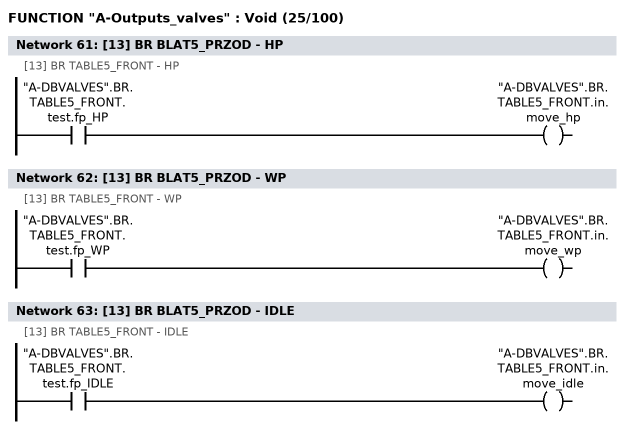
      O "A-DBVALVES".BR.TABLE5_FRONT.test.fp_HP;
//    O     "A-Flags".STATION.IN_HP_STEP
      = "A-DBVALVES".BR.TABLE5_FRONT.in.move_hp;
NETWORK
TITLE = [13] BR BLAT5_PRZOD - WP
//[13] BR TABLE5_FRONT - WP
      O "A-DBVALVES".BR.TABLE5_FRONT.test.fp_WP;
      = "A-DBVALVES".BR.TABLE5_FRONT.in.move_wp;
NETWORK
TITLE = [13] BR BLAT5_PRZOD - IDLE
//[13] BR TABLE5_FRONT - IDLE
      O "A-DBVALVES".BR.TABLE5_FRONT.test.fp_IDLE;
      = "A-DBVALVES".BR.TABLE5_FRONT.in.move_idle;
NETWORK
TITLE = [13] BR BLAT5_PRZOD
//[13] BR TABLE5_FRONT
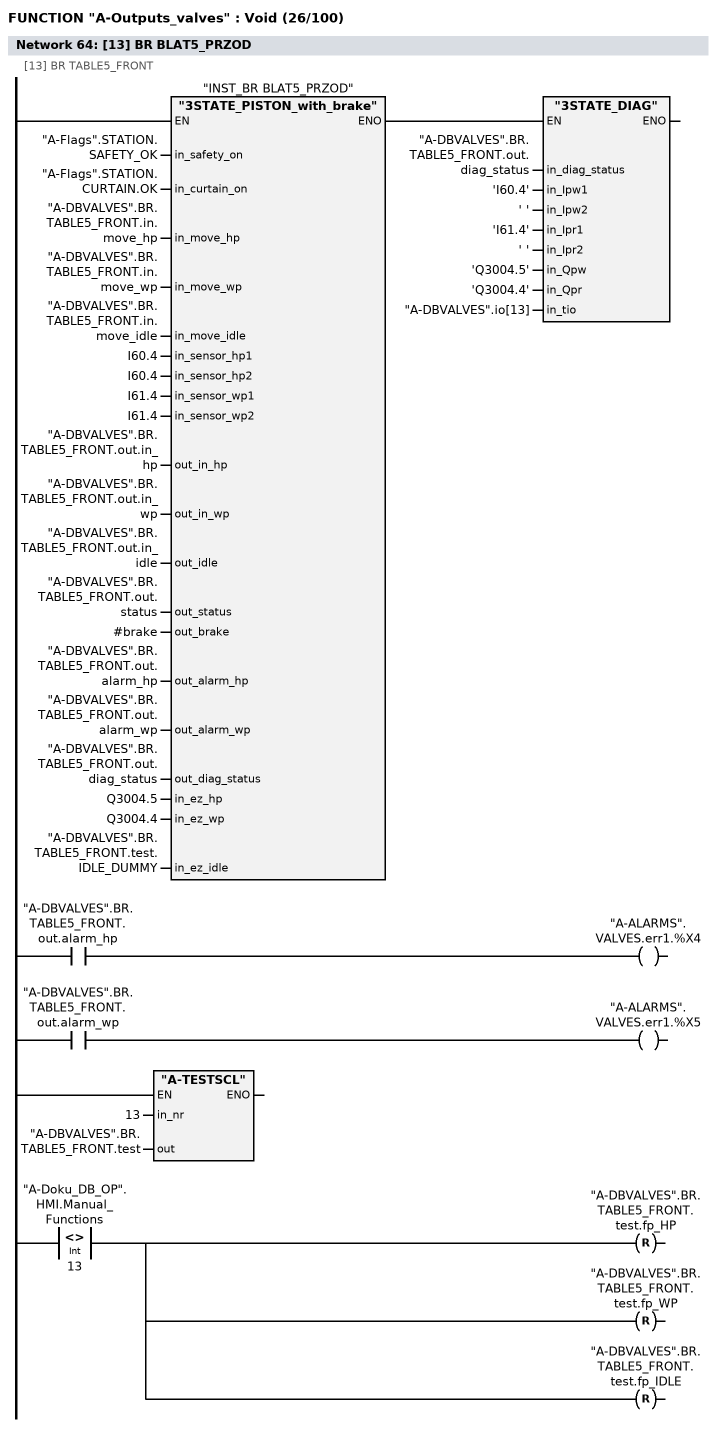
      CALL "3STATE_PISTON_with_brake", "INST_BR BLAT5_PRZOD"
      (  in_safety_on                := "A-Flags".STATION.SAFETY_OK ,
         in_curtain_on               := "A-Flags".STATION.CURTAIN.OK ,
         in_move_hp                  := "A-DBVALVES".BR.TABLE5_FRONT.in.move_hp ,
         in_move_wp                  := "A-DBVALVES".BR.TABLE5_FRONT.in.move_wp ,
         in_move_idle                := "A-DBVALVES".BR.TABLE5_FRONT.in.move_idle ,
         in_sensor_hp1               := I60.4 ,
         in_sensor_hp2               := I60.4 ,
         in_sensor_wp1               := I61.4 ,
         in_sensor_wp2               := I61.4 ,
         out_in_hp                   := "A-DBVALVES".BR.TABLE5_FRONT.out.in_hp ,
         out_in_wp                   := "A-DBVALVES".BR.TABLE5_FRONT.out.in_wp ,
         out_idle                    := "A-DBVALVES".BR.TABLE5_FRONT.out.in_idle ,
         out_status                  := "A-DBVALVES".BR.TABLE5_FRONT.out.status ,
         out_brake                   := #brake ,
         out_alarm_hp                := "A-DBVALVES".BR.TABLE5_FRONT.out.alarm_hp ,
         out_alarm_wp                := "A-DBVALVES".BR.TABLE5_FRONT.out.alarm_wp ,
         out_diag_status             := "A-DBVALVES".BR.TABLE5_FRONT.out.diag_status ,
         in_ez_hp                    := Q3004.5 ,
         in_ez_wp                    := Q3004.4 ,
         in_ez_idle                  := "A-DBVALVES".BR.TABLE5_FRONT.test.IDLE_DUMMY
      );

      CALL "3STATE_DIAG"
      (  in_diag_status              := "A-DBVALVES".BR.TABLE5_FRONT.out.diag_status ,
         in_Ipw1                     := 'I60.4' ,
         in_Ipw2                     := ' ' ,
         in_Ipr1                     := 'I61.4' ,
         in_Ipr2                     := ' ' ,
         in_Qpw                      := 'Q3004.5' ,
         in_Qpr                      := 'Q3004.4' ,
         in_tio                      := "A-DBVALVES".io[13]
      );

      A "A-DBVALVES".BR.TABLE5_FRONT.out.alarm_hp;
      = "A-ALARMS".VALVES.err1.%X4;

      A "A-DBVALVES".BR.TABLE5_FRONT.out.alarm_wp;
      = "A-ALARMS".VALVES.err1.%X5;

      CALL "A-TESTSCL"
      (  in_nr                       := 13 ,
         out                         := "A-DBVALVES".BR.TABLE5_FRONT.test
      );

      A(;
      L "A-Doku_DB_OP".HMI.Manual_Functions;
      L 13;
      <>I;
      );
      R "A-DBVALVES".BR.TABLE5_FRONT.test.fp_HP;
      R "A-DBVALVES".BR.TABLE5_FRONT.test.fp_WP;
      R "A-DBVALVES".BR.TABLE5_FRONT.test.fp_IDLE;
NETWORK
TITLE = -

NETWORK
TITLE = [14] BR BLAT_TYL_LEWY - HP
//[14] BR TABLE_REAR_LEFT - HP
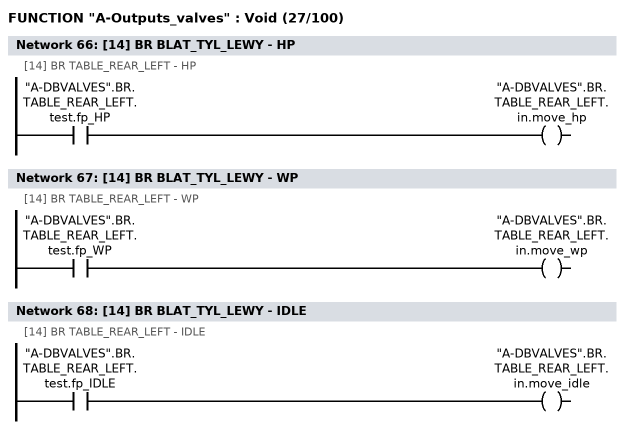
      O "A-DBVALVES".BR.TABLE_REAR_LEFT.test.fp_HP;
//    O     "A-Flags".STATION.IN_HP_STEP
      = "A-DBVALVES".BR.TABLE_REAR_LEFT.in.move_hp;
NETWORK
TITLE = [14] BR BLAT_TYL_LEWY - WP
//[14] BR TABLE_REAR_LEFT - WP
      O "A-DBVALVES".BR.TABLE_REAR_LEFT.test.fp_WP;
      = "A-DBVALVES".BR.TABLE_REAR_LEFT.in.move_wp;
NETWORK
TITLE = [14] BR BLAT_TYL_LEWY - IDLE
//[14] BR TABLE_REAR_LEFT - IDLE
      O "A-DBVALVES".BR.TABLE_REAR_LEFT.test.fp_IDLE;
      = "A-DBVALVES".BR.TABLE_REAR_LEFT.in.move_idle;
NETWORK
TITLE = [14] BR BLAT_TYL_LEWY
//[14] BR TABLE_REAR_LEFT
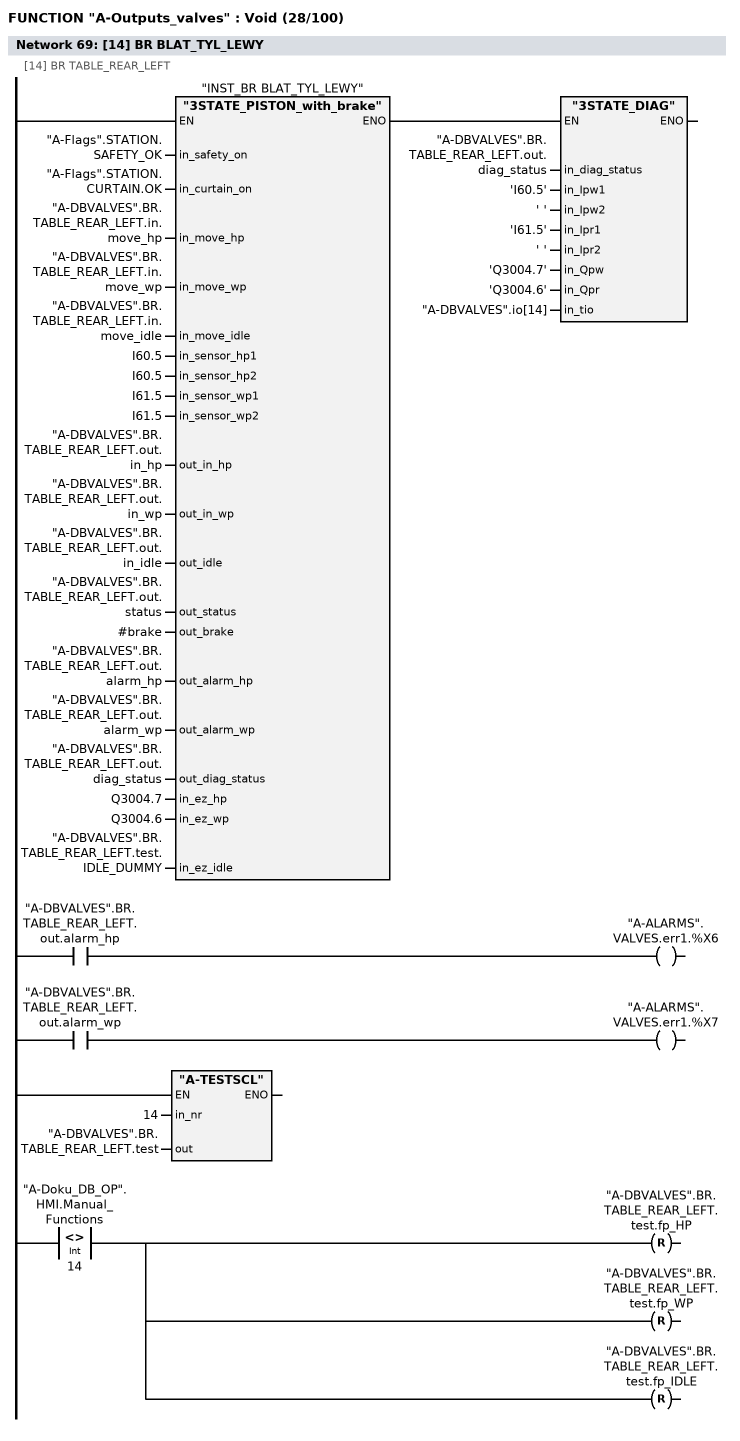
      CALL "3STATE_PISTON_with_brake", "INST_BR BLAT_TYL_LEWY"
      (  in_safety_on                := "A-Flags".STATION.SAFETY_OK ,
         in_curtain_on               := "A-Flags".STATION.CURTAIN.OK ,
         in_move_hp                  := "A-DBVALVES".BR.TABLE_REAR_LEFT.in.move_hp ,
         in_move_wp                  := "A-DBVALVES".BR.TABLE_REAR_LEFT.in.move_wp ,
         in_move_idle                := "A-DBVALVES".BR.TABLE_REAR_LEFT.in.move_idle ,
         in_sensor_hp1               := I60.5 ,
         in_sensor_hp2               := I60.5 ,
         in_sensor_wp1               := I61.5 ,
         in_sensor_wp2               := I61.5 ,
         out_in_hp                   := "A-DBVALVES".BR.TABLE_REAR_LEFT.out.in_hp ,
         out_in_wp                   := "A-DBVALVES".BR.TABLE_REAR_LEFT.out.in_wp ,
         out_idle                    := "A-DBVALVES".BR.TABLE_REAR_LEFT.out.in_idle ,
         out_status                  := "A-DBVALVES".BR.TABLE_REAR_LEFT.out.status ,
         out_brake                   := #brake ,
         out_alarm_hp                := "A-DBVALVES".BR.TABLE_REAR_LEFT.out.alarm_hp ,
         out_alarm_wp                := "A-DBVALVES".BR.TABLE_REAR_LEFT.out.alarm_wp ,
         out_diag_status             := "A-DBVALVES".BR.TABLE_REAR_LEFT.out.diag_status ,
         in_ez_hp                    := Q3004.7 ,
         in_ez_wp                    := Q3004.6 ,
         in_ez_idle                  := "A-DBVALVES".BR.TABLE_REAR_LEFT.test.IDLE_DUMMY
      );

      CALL "3STATE_DIAG"
      (  in_diag_status              := "A-DBVALVES".BR.TABLE_REAR_LEFT.out.diag_status ,
         in_Ipw1                     := 'I60.5' ,
         in_Ipw2                     := ' ' ,
         in_Ipr1                     := 'I61.5' ,
         in_Ipr2                     := ' ' ,
         in_Qpw                      := 'Q3004.7' ,
         in_Qpr                      := 'Q3004.6' ,
         in_tio                      := "A-DBVALVES".io[14]
      );

      A "A-DBVALVES".BR.TABLE_REAR_LEFT.out.alarm_hp;
      = "A-ALARMS".VALVES.err1.%X6;

      A "A-DBVALVES".BR.TABLE_REAR_LEFT.out.alarm_wp;
      = "A-ALARMS".VALVES.err1.%X7;

      CALL "A-TESTSCL"
      (  in_nr                       := 14 ,
         out                         := "A-DBVALVES".BR.TABLE_REAR_LEFT.test
      );

      A(;
      L "A-Doku_DB_OP".HMI.Manual_Functions;
      L 14;
      <>I;
      );
      R "A-DBVALVES".BR.TABLE_REAR_LEFT.test.fp_HP;
      R "A-DBVALVES".BR.TABLE_REAR_LEFT.test.fp_WP;
      R "A-DBVALVES".BR.TABLE_REAR_LEFT.test.fp_IDLE;
NETWORK
TITLE = -

NETWORK
TITLE = [15] BR BLAT_TYL_PRAWY - HP
//[15] BR TABLE_REAR_RIGHT - HP
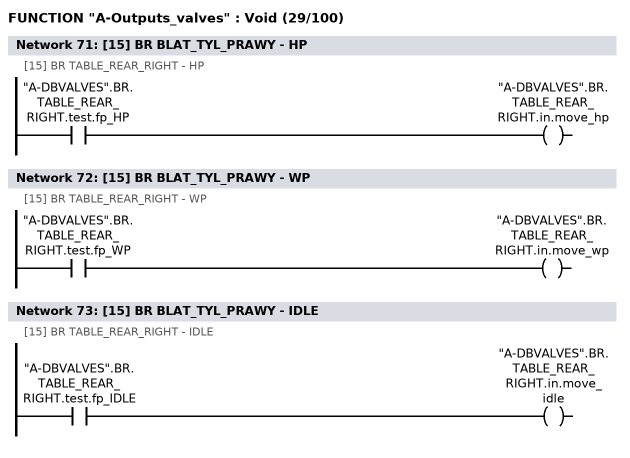
      O "A-DBVALVES".BR.TABLE_REAR_RIGHT.test.fp_HP;
//    O     "A-Flags".STATION.IN_HP_STEP
      = "A-DBVALVES".BR.TABLE_REAR_RIGHT.in.move_hp;
NETWORK
TITLE = [15] BR BLAT_TYL_PRAWY - WP
//[15] BR TABLE_REAR_RIGHT - WP
      O "A-DBVALVES".BR.TABLE_REAR_RIGHT.test.fp_WP;
      = "A-DBVALVES".BR.TABLE_REAR_RIGHT.in.move_wp;
NETWORK
TITLE = [15] BR BLAT_TYL_PRAWY - IDLE
//[15] BR TABLE_REAR_RIGHT - IDLE
      O "A-DBVALVES".BR.TABLE_REAR_RIGHT.test.fp_IDLE;
      = "A-DBVALVES".BR.TABLE_REAR_RIGHT.in.move_idle;
NETWORK
TITLE = [15] BR BLAT_TYL_PRAWY
//[15] BR TABLE_REAR_RIGHT
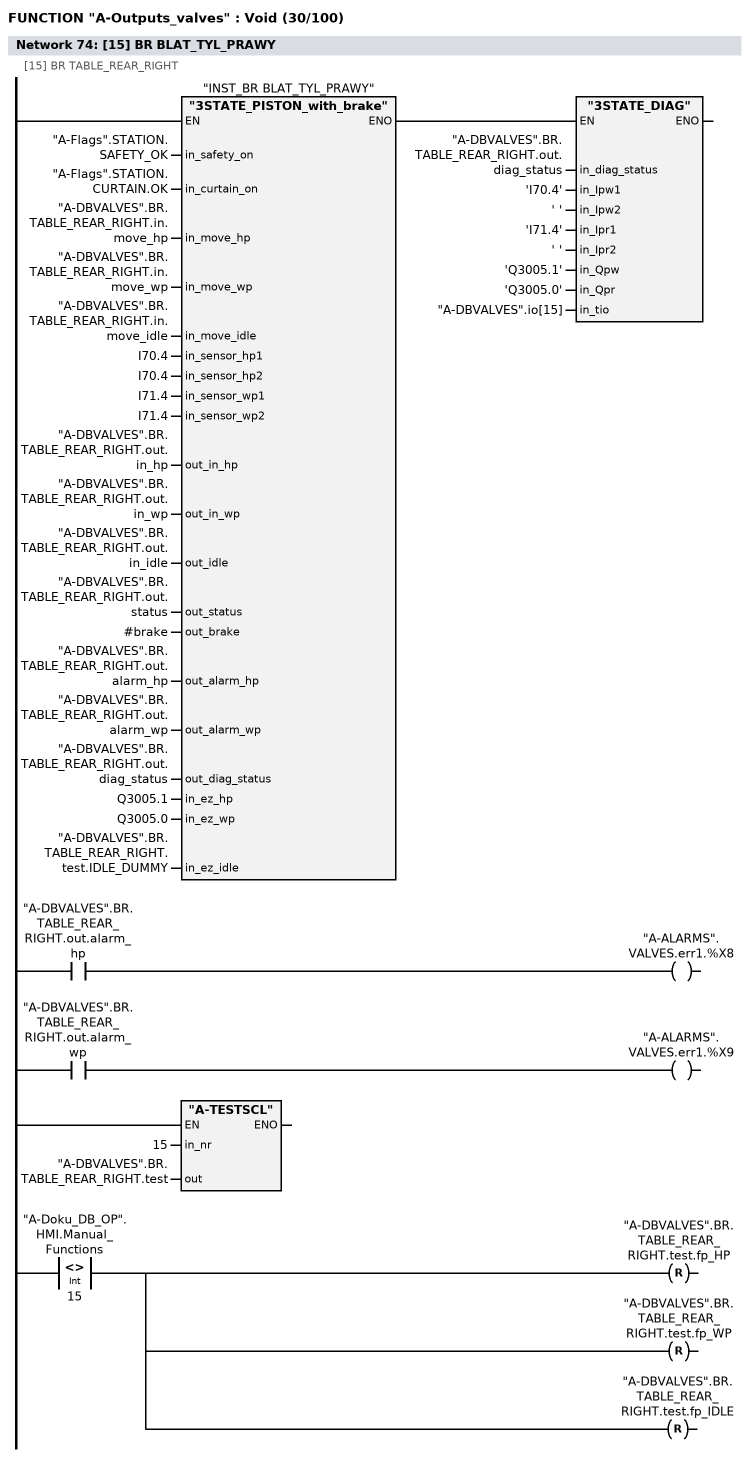
      CALL "3STATE_PISTON_with_brake", "INST_BR BLAT_TYL_PRAWY"
      (  in_safety_on                := "A-Flags".STATION.SAFETY_OK ,
         in_curtain_on               := "A-Flags".STATION.CURTAIN.OK ,
         in_move_hp                  := "A-DBVALVES".BR.TABLE_REAR_RIGHT.in.move_hp ,
         in_move_wp                  := "A-DBVALVES".BR.TABLE_REAR_RIGHT.in.move_wp ,
         in_move_idle                := "A-DBVALVES".BR.TABLE_REAR_RIGHT.in.move_idle ,
         in_sensor_hp1               := I70.4 ,
         in_sensor_hp2               := I70.4 ,
         in_sensor_wp1               := I71.4 ,
         in_sensor_wp2               := I71.4 ,
         out_in_hp                   := "A-DBVALVES".BR.TABLE_REAR_RIGHT.out.in_hp ,
         out_in_wp                   := "A-DBVALVES".BR.TABLE_REAR_RIGHT.out.in_wp ,
         out_idle                    := "A-DBVALVES".BR.TABLE_REAR_RIGHT.out.in_idle ,
         out_status                  := "A-DBVALVES".BR.TABLE_REAR_RIGHT.out.status ,
         out_brake                   := #brake ,
         out_alarm_hp                := "A-DBVALVES".BR.TABLE_REAR_RIGHT.out.alarm_hp ,
         out_alarm_wp                := "A-DBVALVES".BR.TABLE_REAR_RIGHT.out.alarm_wp ,
         out_diag_status             := "A-DBVALVES".BR.TABLE_REAR_RIGHT.out.diag_status ,
         in_ez_hp                    := Q3005.1 ,
         in_ez_wp                    := Q3005.0 ,
         in_ez_idle                  := "A-DBVALVES".BR.TABLE_REAR_RIGHT.test.IDLE_DUMMY
      );

      CALL "3STATE_DIAG"
      (  in_diag_status              := "A-DBVALVES".BR.TABLE_REAR_RIGHT.out.diag_status ,
         in_Ipw1                     := 'I70.4' ,
         in_Ipw2                     := ' ' ,
         in_Ipr1                     := 'I71.4' ,
         in_Ipr2                     := ' ' ,
         in_Qpw                      := 'Q3005.1' ,
         in_Qpr                      := 'Q3005.0' ,
         in_tio                      := "A-DBVALVES".io[15]
      );

      A "A-DBVALVES".BR.TABLE_REAR_RIGHT.out.alarm_hp;
      = "A-ALARMS".VALVES.err1.%X8;

      A "A-DBVALVES".BR.TABLE_REAR_RIGHT.out.alarm_wp;
      = "A-ALARMS".VALVES.err1.%X9;

      CALL "A-TESTSCL"
      (  in_nr                       := 15 ,
         out                         := "A-DBVALVES".BR.TABLE_REAR_RIGHT.test
      );

      A(;
      L "A-Doku_DB_OP".HMI.Manual_Functions;
      L 15;
      <>I;
      );
      R "A-DBVALVES".BR.TABLE_REAR_RIGHT.test.fp_HP;
      R "A-DBVALVES".BR.TABLE_REAR_RIGHT.test.fp_WP;
      R "A-DBVALVES".BR.TABLE_REAR_RIGHT.test.fp_IDLE;
NETWORK
TITLE = -

NETWORK
TITLE = [16] ST1 PRZESUW_STACJI - HP
//[16] ST1 STATION_MOVEMENT - HP
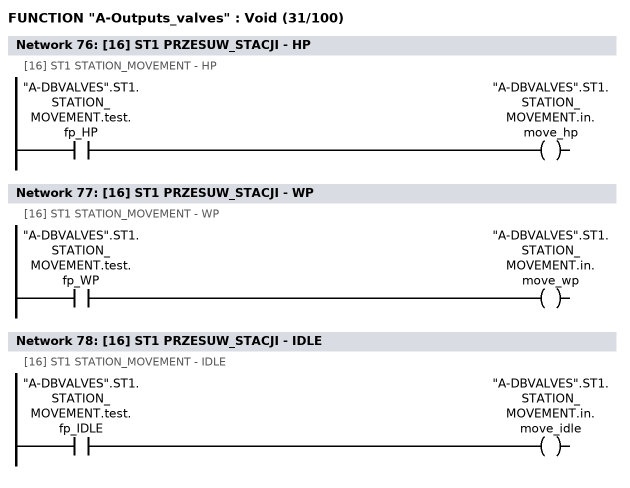
      O "A-DBVALVES".ST1.STATION_MOVEMENT.test.fp_HP;
//    O     "A-Flags".STATION.IN_HP_STEP
      = "A-DBVALVES".ST1.STATION_MOVEMENT.in.move_hp;
NETWORK
TITLE = [16] ST1 PRZESUW_STACJI - WP
//[16] ST1 STATION_MOVEMENT - WP
      O "A-DBVALVES".ST1.STATION_MOVEMENT.test.fp_WP;
      = "A-DBVALVES".ST1.STATION_MOVEMENT.in.move_wp;
NETWORK
TITLE = [16] ST1 PRZESUW_STACJI - IDLE
//[16] ST1 STATION_MOVEMENT - IDLE
      O "A-DBVALVES".ST1.STATION_MOVEMENT.test.fp_IDLE;
      = "A-DBVALVES".ST1.STATION_MOVEMENT.in.move_idle;
NETWORK
TITLE = [16] ST1 PRZESUW_STACJI
//[16] ST1 STATION_MOVEMENT
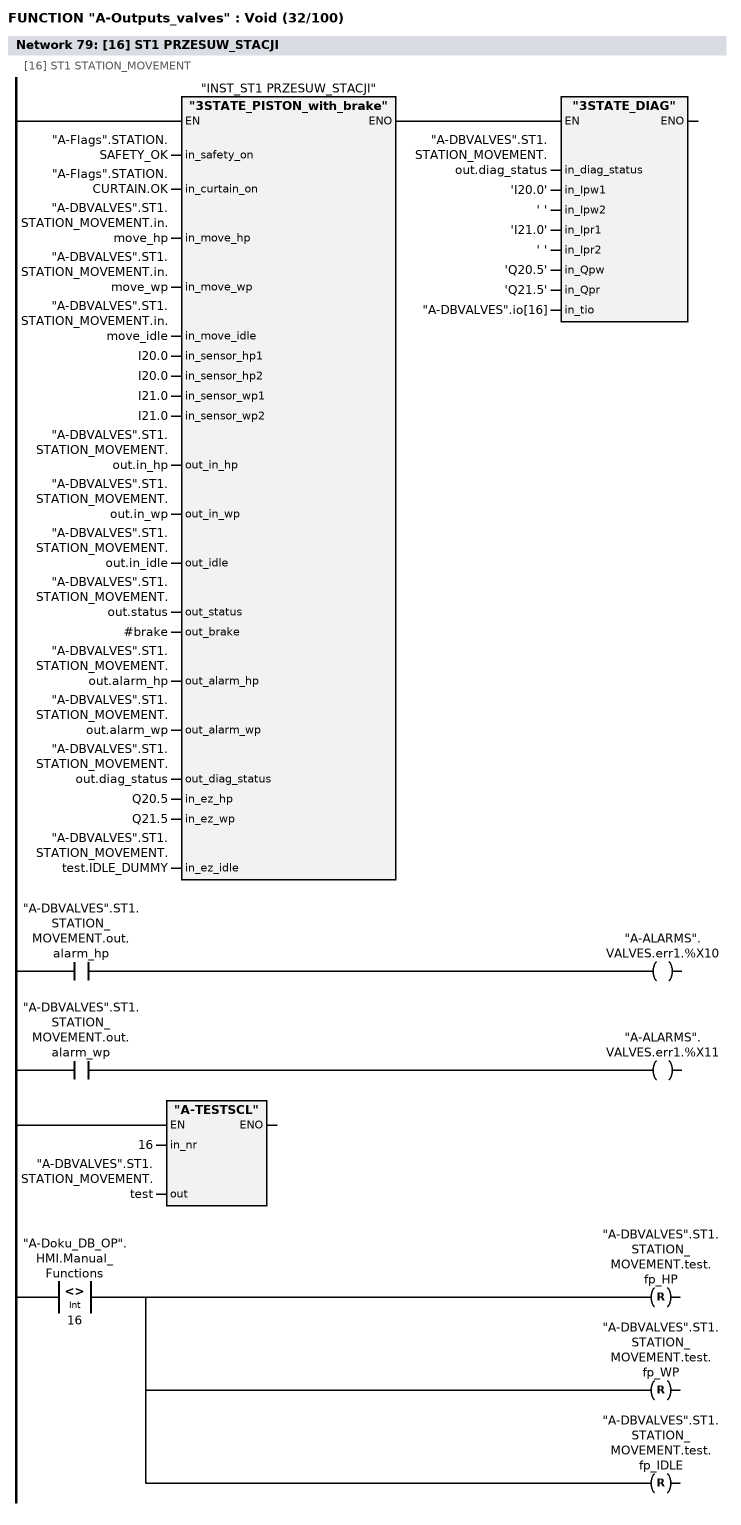
      CALL "3STATE_PISTON_with_brake", "INST_ST1 PRZESUW_STACJI"
      (  in_safety_on                := "A-Flags".STATION.SAFETY_OK ,
         in_curtain_on               := "A-Flags".STATION.CURTAIN.OK ,
         in_move_hp                  := "A-DBVALVES".ST1.STATION_MOVEMENT.in.move_hp ,
         in_move_wp                  := "A-DBVALVES".ST1.STATION_MOVEMENT.in.move_wp ,
         in_move_idle                := "A-DBVALVES".ST1.STATION_MOVEMENT.in.move_idle ,
         in_sensor_hp1               := I20.0 ,
         in_sensor_hp2               := I20.0 ,
         in_sensor_wp1               := I21.0 ,
         in_sensor_wp2               := I21.0 ,
         out_in_hp                   := "A-DBVALVES".ST1.STATION_MOVEMENT.out.in_hp ,
         out_in_wp                   := "A-DBVALVES".ST1.STATION_MOVEMENT.out.in_wp ,
         out_idle                    := "A-DBVALVES".ST1.STATION_MOVEMENT.out.in_idle ,
         out_status                  := "A-DBVALVES".ST1.STATION_MOVEMENT.out.status ,
         out_brake                   := #brake ,
         out_alarm_hp                := "A-DBVALVES".ST1.STATION_MOVEMENT.out.alarm_hp ,
         out_alarm_wp                := "A-DBVALVES".ST1.STATION_MOVEMENT.out.alarm_wp ,
         out_diag_status             := "A-DBVALVES".ST1.STATION_MOVEMENT.out.diag_status ,
         in_ez_hp                    := Q20.5 ,
         in_ez_wp                    := Q21.5 ,
         in_ez_idle                  := "A-DBVALVES".ST1.STATION_MOVEMENT.test.IDLE_DUMMY
      );

      CALL "3STATE_DIAG"
      (  in_diag_status              := "A-DBVALVES".ST1.STATION_MOVEMENT.out.diag_status ,
         in_Ipw1                     := 'I20.0' ,
         in_Ipw2                     := ' ' ,
         in_Ipr1                     := 'I21.0' ,
         in_Ipr2                     := ' ' ,
         in_Qpw                      := 'Q20.5' ,
         in_Qpr                      := 'Q21.5' ,
         in_tio                      := "A-DBVALVES".io[16]
      );

      A "A-DBVALVES".ST1.STATION_MOVEMENT.out.alarm_hp;
      = "A-ALARMS".VALVES.err1.%X10;

      A "A-DBVALVES".ST1.STATION_MOVEMENT.out.alarm_wp;
      = "A-ALARMS".VALVES.err1.%X11;

      CALL "A-TESTSCL"
      (  in_nr                       := 16 ,
         out                         := "A-DBVALVES".ST1.STATION_MOVEMENT.test
      );

      A(;
      L "A-Doku_DB_OP".HMI.Manual_Functions;
      L 16;
      <>I;
      );
      R "A-DBVALVES".ST1.STATION_MOVEMENT.test.fp_HP;
      R "A-DBVALVES".ST1.STATION_MOVEMENT.test.fp_WP;
      R "A-DBVALVES".ST1.STATION_MOVEMENT.test.fp_IDLE;
NETWORK
TITLE = -

NETWORK
TITLE = [17] ST1 WYSUW_MIECZA - HP
//[17] ST1 SWORD_SLIDE_OUT - HP
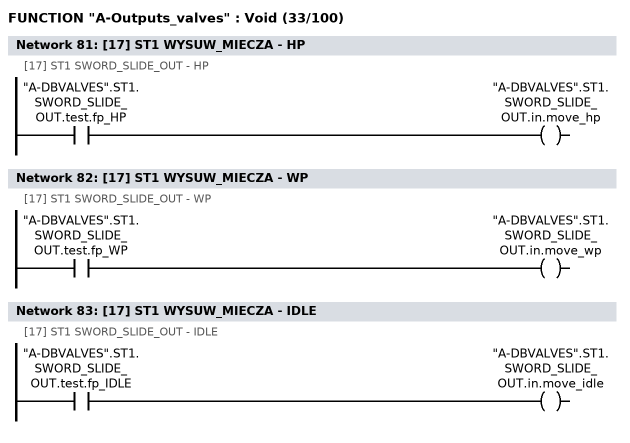
      O "A-DBVALVES".ST1.SWORD_SLIDE_OUT.test.fp_HP;
//    O     "A-Flags".STATION.IN_HP_STEP
      = "A-DBVALVES".ST1.SWORD_SLIDE_OUT.in.move_hp;
NETWORK
TITLE = [17] ST1 WYSUW_MIECZA - WP
//[17] ST1 SWORD_SLIDE_OUT - WP
      O "A-DBVALVES".ST1.SWORD_SLIDE_OUT.test.fp_WP;
      = "A-DBVALVES".ST1.SWORD_SLIDE_OUT.in.move_wp;
NETWORK
TITLE = [17] ST1 WYSUW_MIECZA - IDLE
//[17] ST1 SWORD_SLIDE_OUT - IDLE
      O "A-DBVALVES".ST1.SWORD_SLIDE_OUT.test.fp_IDLE;
      = "A-DBVALVES".ST1.SWORD_SLIDE_OUT.in.move_idle;
NETWORK
TITLE = [17] ST1 WYSUW_MIECZA
//[17] ST1 SWORD_SLIDE_OUT
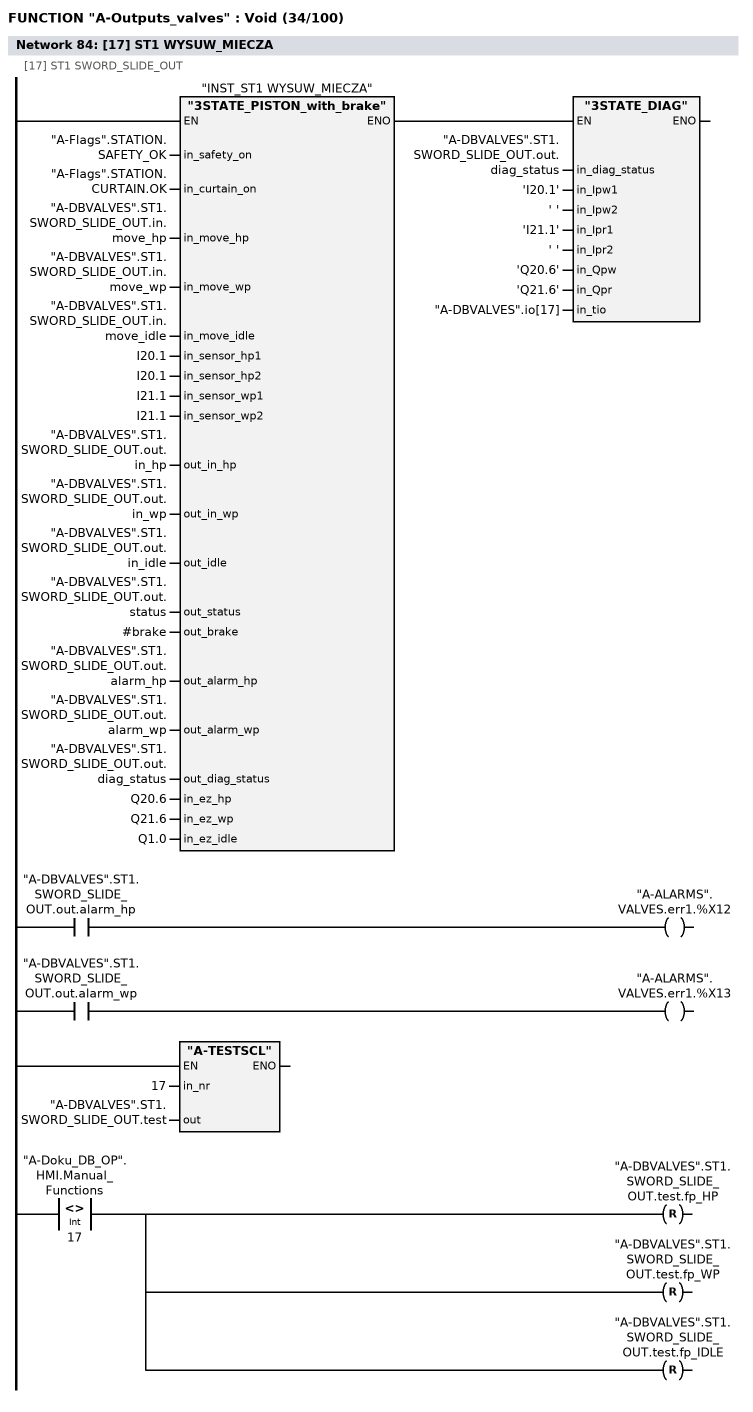
      CALL "3STATE_PISTON_with_brake", "INST_ST1 WYSUW_MIECZA"
      (  in_safety_on                := "A-Flags".STATION.SAFETY_OK ,
         in_curtain_on               := "A-Flags".STATION.CURTAIN.OK ,
         in_move_hp                  := "A-DBVALVES".ST1.SWORD_SLIDE_OUT.in.move_hp ,
         in_move_wp                  := "A-DBVALVES".ST1.SWORD_SLIDE_OUT.in.move_wp ,
         in_move_idle                := "A-DBVALVES".ST1.SWORD_SLIDE_OUT.in.move_idle ,
         in_sensor_hp1               := I20.1 ,
         in_sensor_hp2               := I20.1 ,
         in_sensor_wp1               := I21.1 ,
         in_sensor_wp2               := I21.1 ,
         out_in_hp                   := "A-DBVALVES".ST1.SWORD_SLIDE_OUT.out.in_hp ,
         out_in_wp                   := "A-DBVALVES".ST1.SWORD_SLIDE_OUT.out.in_wp ,
         out_idle                    := "A-DBVALVES".ST1.SWORD_SLIDE_OUT.out.in_idle ,
         out_status                  := "A-DBVALVES".ST1.SWORD_SLIDE_OUT.out.status ,
         out_brake                   := #brake ,
         out_alarm_hp                := "A-DBVALVES".ST1.SWORD_SLIDE_OUT.out.alarm_hp ,
         out_alarm_wp                := "A-DBVALVES".ST1.SWORD_SLIDE_OUT.out.alarm_wp ,
         out_diag_status             := "A-DBVALVES".ST1.SWORD_SLIDE_OUT.out.diag_status ,
         in_ez_hp                    := Q20.6 ,
         in_ez_wp                    := Q21.6 ,
         in_ez_idle                  := Q1.0
      );

      CALL "3STATE_DIAG"
      (  in_diag_status              := "A-DBVALVES".ST1.SWORD_SLIDE_OUT.out.diag_status ,
         in_Ipw1                     := 'I20.1' ,
         in_Ipw2                     := ' ' ,
         in_Ipr1                     := 'I21.1' ,
         in_Ipr2                     := ' ' ,
         in_Qpw                      := 'Q20.6' ,
         in_Qpr                      := 'Q21.6' ,
         in_tio                      := "A-DBVALVES".io[17]
      );

      A "A-DBVALVES".ST1.SWORD_SLIDE_OUT.out.alarm_hp;
      = "A-ALARMS".VALVES.err1.%X12;

      A "A-DBVALVES".ST1.SWORD_SLIDE_OUT.out.alarm_wp;
      = "A-ALARMS".VALVES.err1.%X13;

      CALL "A-TESTSCL"
      (  in_nr                       := 17 ,
         out                         := "A-DBVALVES".ST1.SWORD_SLIDE_OUT.test
      );

      A(;
      L "A-Doku_DB_OP".HMI.Manual_Functions;
      L 17;
      <>I;
      );
      R "A-DBVALVES".ST1.SWORD_SLIDE_OUT.test.fp_HP;
      R "A-DBVALVES".ST1.SWORD_SLIDE_OUT.test.fp_WP;
      R "A-DBVALVES".ST1.SWORD_SLIDE_OUT.test.fp_IDLE;
NETWORK
TITLE = -

NETWORK
TITLE = [18] ST1 MIECZ - HP
//[18] ST1 SWORD - HP
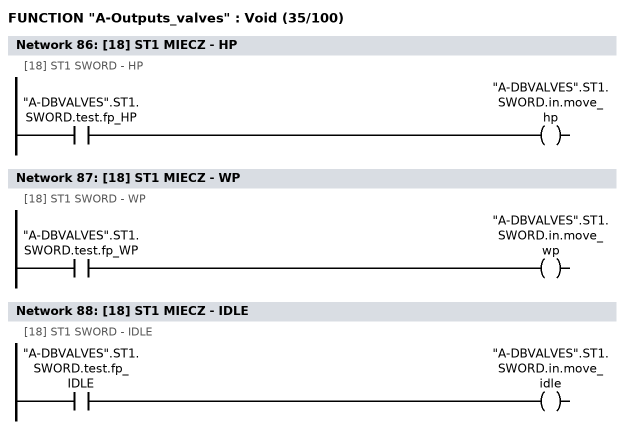
      O "A-DBVALVES".ST1.SWORD.test.fp_HP;
//    O     "A-Flags".STATION.IN_HP_STEP
      = "A-DBVALVES".ST1.SWORD.in.move_hp;
NETWORK
TITLE = [18] ST1 MIECZ - WP
//[18] ST1 SWORD - WP
      O "A-DBVALVES".ST1.SWORD.test.fp_WP;
      = "A-DBVALVES".ST1.SWORD.in.move_wp;
NETWORK
TITLE = [18] ST1 MIECZ - IDLE
//[18] ST1 SWORD - IDLE
      O "A-DBVALVES".ST1.SWORD.test.fp_IDLE;
      = "A-DBVALVES".ST1.SWORD.in.move_idle;
NETWORK
TITLE = [18] ST1 MIECZ
//[18] ST1 SWORD
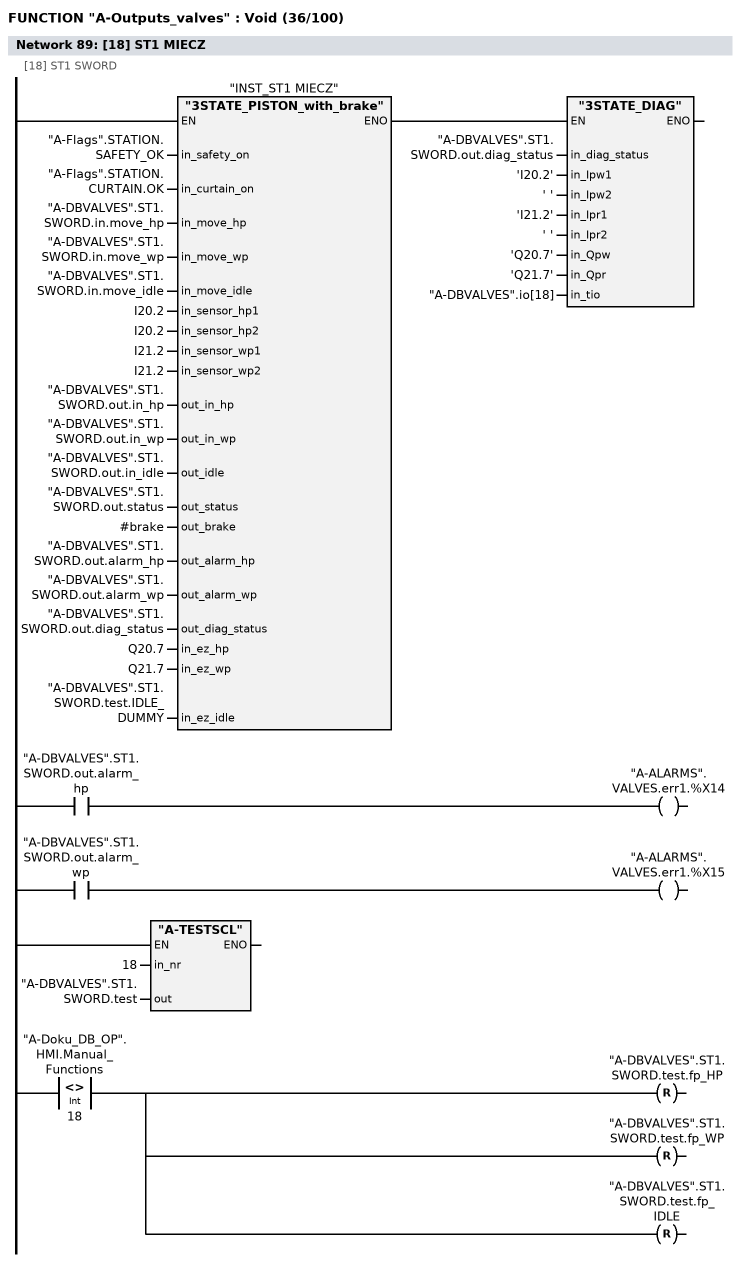
      CALL "3STATE_PISTON_with_brake", "INST_ST1 MIECZ"
      (  in_safety_on                := "A-Flags".STATION.SAFETY_OK ,
         in_curtain_on               := "A-Flags".STATION.CURTAIN.OK ,
         in_move_hp                  := "A-DBVALVES".ST1.SWORD.in.move_hp ,
         in_move_wp                  := "A-DBVALVES".ST1.SWORD.in.move_wp ,
         in_move_idle                := "A-DBVALVES".ST1.SWORD.in.move_idle ,
         in_sensor_hp1               := I20.2 ,
         in_sensor_hp2               := I20.2 ,
         in_sensor_wp1               := I21.2 ,
         in_sensor_wp2               := I21.2 ,
         out_in_hp                   := "A-DBVALVES".ST1.SWORD.out.in_hp ,
         out_in_wp                   := "A-DBVALVES".ST1.SWORD.out.in_wp ,
         out_idle                    := "A-DBVALVES".ST1.SWORD.out.in_idle ,
         out_status                  := "A-DBVALVES".ST1.SWORD.out.status ,
         out_brake                   := #brake ,
         out_alarm_hp                := "A-DBVALVES".ST1.SWORD.out.alarm_hp ,
         out_alarm_wp                := "A-DBVALVES".ST1.SWORD.out.alarm_wp ,
         out_diag_status             := "A-DBVALVES".ST1.SWORD.out.diag_status ,
         in_ez_hp                    := Q20.7 ,
         in_ez_wp                    := Q21.7 ,
         in_ez_idle                  := "A-DBVALVES".ST1.SWORD.test.IDLE_DUMMY
      );

      CALL "3STATE_DIAG"
      (  in_diag_status              := "A-DBVALVES".ST1.SWORD.out.diag_status ,
         in_Ipw1                     := 'I20.2' ,
         in_Ipw2                     := ' ' ,
         in_Ipr1                     := 'I21.2' ,
         in_Ipr2                     := ' ' ,
         in_Qpw                      := 'Q20.7' ,
         in_Qpr                      := 'Q21.7' ,
         in_tio                      := "A-DBVALVES".io[18]
      );

      A "A-DBVALVES".ST1.SWORD.out.alarm_hp;
      = "A-ALARMS".VALVES.err1.%X14;

      A "A-DBVALVES".ST1.SWORD.out.alarm_wp;
      = "A-ALARMS".VALVES.err1.%X15;

      CALL "A-TESTSCL"
      (  in_nr                       := 18 ,
         out                         := "A-DBVALVES".ST1.SWORD.test
      );

      A(;
      L "A-Doku_DB_OP".HMI.Manual_Functions;
      L 18;
      <>I;
      );
      R "A-DBVALVES".ST1.SWORD.test.fp_HP;
      R "A-DBVALVES".ST1.SWORD.test.fp_WP;
      R "A-DBVALVES".ST1.SWORD.test.fp_IDLE;
NETWORK
TITLE = -

NETWORK
TITLE = [19] ST2 PRZESUW_STACJI - HP
//[19] ST2 STATION_MOVEMENT - HP
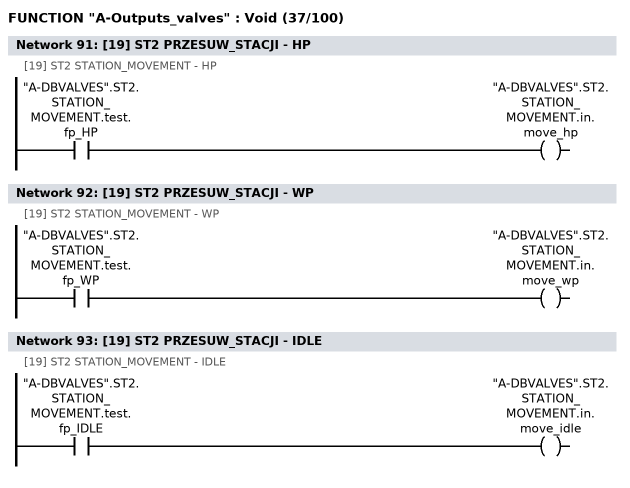
      O "A-DBVALVES".ST2.STATION_MOVEMENT.test.fp_HP;
//    O     "A-Flags".STATION.IN_HP_STEP
      = "A-DBVALVES".ST2.STATION_MOVEMENT.in.move_hp;
NETWORK
TITLE = [19] ST2 PRZESUW_STACJI - WP
//[19] ST2 STATION_MOVEMENT - WP
      O "A-DBVALVES".ST2.STATION_MOVEMENT.test.fp_WP;
      = "A-DBVALVES".ST2.STATION_MOVEMENT.in.move_wp;
NETWORK
TITLE = [19] ST2 PRZESUW_STACJI - IDLE
//[19] ST2 STATION_MOVEMENT - IDLE
      O "A-DBVALVES".ST2.STATION_MOVEMENT.test.fp_IDLE;
      = "A-DBVALVES".ST2.STATION_MOVEMENT.in.move_idle;
NETWORK
TITLE = [19] ST2 PRZESUW_STACJI
//[19] ST2 STATION_MOVEMENT
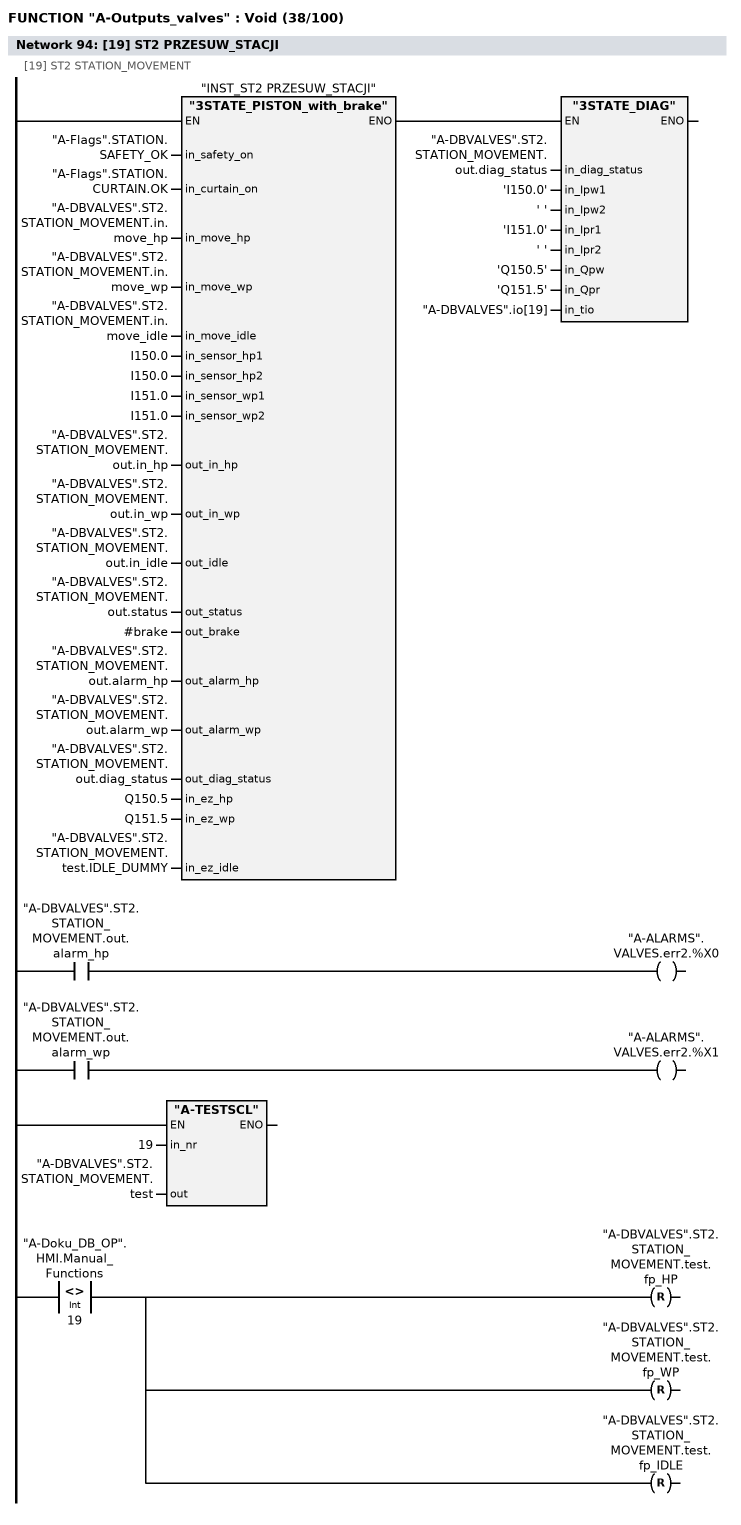
      CALL "3STATE_PISTON_with_brake", "INST_ST2 PRZESUW_STACJI"
      (  in_safety_on                := "A-Flags".STATION.SAFETY_OK ,
         in_curtain_on               := "A-Flags".STATION.CURTAIN.OK ,
         in_move_hp                  := "A-DBVALVES".ST2.STATION_MOVEMENT.in.move_hp ,
         in_move_wp                  := "A-DBVALVES".ST2.STATION_MOVEMENT.in.move_wp ,
         in_move_idle                := "A-DBVALVES".ST2.STATION_MOVEMENT.in.move_idle ,
         in_sensor_hp1               := I150.0 ,
         in_sensor_hp2               := I150.0 ,
         in_sensor_wp1               := I151.0 ,
         in_sensor_wp2               := I151.0 ,
         out_in_hp                   := "A-DBVALVES".ST2.STATION_MOVEMENT.out.in_hp ,
         out_in_wp                   := "A-DBVALVES".ST2.STATION_MOVEMENT.out.in_wp ,
         out_idle                    := "A-DBVALVES".ST2.STATION_MOVEMENT.out.in_idle ,
         out_status                  := "A-DBVALVES".ST2.STATION_MOVEMENT.out.status ,
         out_brake                   := #brake ,
         out_alarm_hp                := "A-DBVALVES".ST2.STATION_MOVEMENT.out.alarm_hp ,
         out_alarm_wp                := "A-DBVALVES".ST2.STATION_MOVEMENT.out.alarm_wp ,
         out_diag_status             := "A-DBVALVES".ST2.STATION_MOVEMENT.out.diag_status ,
         in_ez_hp                    := Q150.5 ,
         in_ez_wp                    := Q151.5 ,
         in_ez_idle                  := "A-DBVALVES".ST2.STATION_MOVEMENT.test.IDLE_DUMMY
      );

      CALL "3STATE_DIAG"
      (  in_diag_status              := "A-DBVALVES".ST2.STATION_MOVEMENT.out.diag_status ,
         in_Ipw1                     := 'I150.0' ,
         in_Ipw2                     := ' ' ,
         in_Ipr1                     := 'I151.0' ,
         in_Ipr2                     := ' ' ,
         in_Qpw                      := 'Q150.5' ,
         in_Qpr                      := 'Q151.5' ,
         in_tio                      := "A-DBVALVES".io[19]
      );

      A "A-DBVALVES".ST2.STATION_MOVEMENT.out.alarm_hp;
      = "A-ALARMS".VALVES.err2.%X0;

      A "A-DBVALVES".ST2.STATION_MOVEMENT.out.alarm_wp;
      = "A-ALARMS".VALVES.err2.%X1;

      CALL "A-TESTSCL"
      (  in_nr                       := 19 ,
         out                         := "A-DBVALVES".ST2.STATION_MOVEMENT.test
      );

      A(;
      L "A-Doku_DB_OP".HMI.Manual_Functions;
      L 19;
      <>I;
      );
      R "A-DBVALVES".ST2.STATION_MOVEMENT.test.fp_HP;
      R "A-DBVALVES".ST2.STATION_MOVEMENT.test.fp_WP;
      R "A-DBVALVES".ST2.STATION_MOVEMENT.test.fp_IDLE;
NETWORK
TITLE = -

NETWORK
TITLE = [20] ST2 WYSUW_MIECZA - HP
//[20] ST2 SWORD_SLIDE_OUT - HP
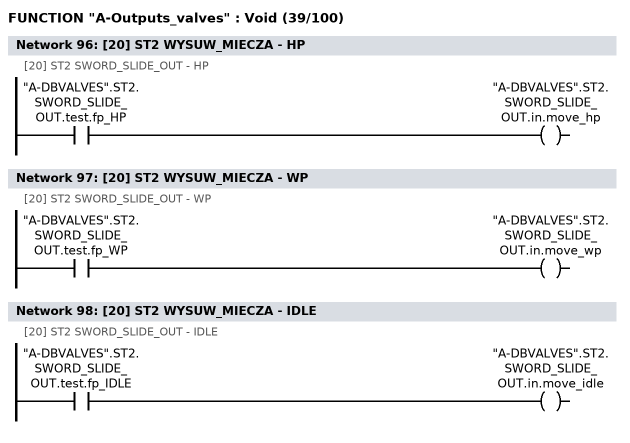
      O "A-DBVALVES".ST2.SWORD_SLIDE_OUT.test.fp_HP;
//    O     "A-Flags".STATION.IN_HP_STEP
      = "A-DBVALVES".ST2.SWORD_SLIDE_OUT.in.move_hp;
NETWORK
TITLE = [20] ST2 WYSUW_MIECZA - WP
//[20] ST2 SWORD_SLIDE_OUT - WP
      O "A-DBVALVES".ST2.SWORD_SLIDE_OUT.test.fp_WP;
      = "A-DBVALVES".ST2.SWORD_SLIDE_OUT.in.move_wp;
NETWORK
TITLE = [20] ST2 WYSUW_MIECZA - IDLE
//[20] ST2 SWORD_SLIDE_OUT - IDLE
      O "A-DBVALVES".ST2.SWORD_SLIDE_OUT.test.fp_IDLE;
      = "A-DBVALVES".ST2.SWORD_SLIDE_OUT.in.move_idle;
NETWORK
TITLE = [20] ST2 WYSUW_MIECZA
//[20] ST2 SWORD_SLIDE_OUT
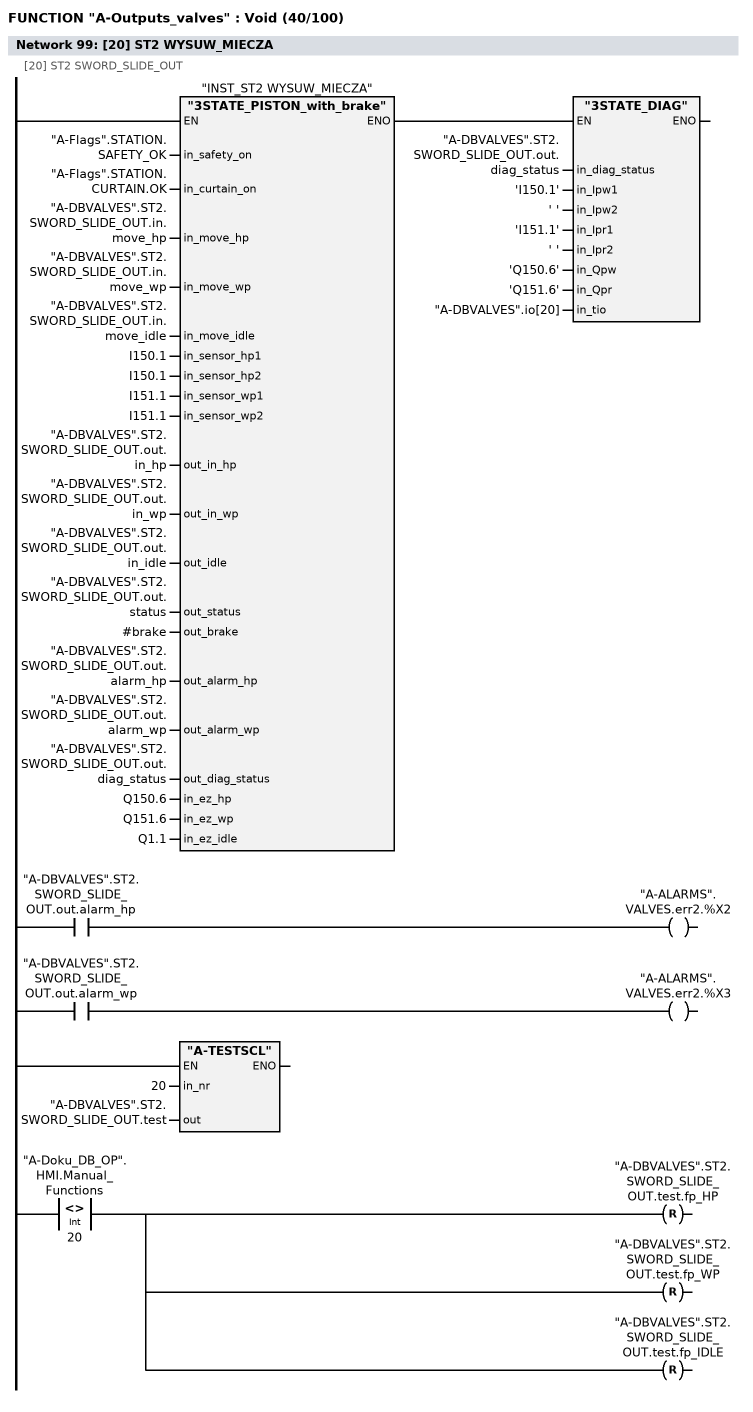
      CALL "3STATE_PISTON_with_brake", "INST_ST2 WYSUW_MIECZA"
      (  in_safety_on                := "A-Flags".STATION.SAFETY_OK ,
         in_curtain_on               := "A-Flags".STATION.CURTAIN.OK ,
         in_move_hp                  := "A-DBVALVES".ST2.SWORD_SLIDE_OUT.in.move_hp ,
         in_move_wp                  := "A-DBVALVES".ST2.SWORD_SLIDE_OUT.in.move_wp ,
         in_move_idle                := "A-DBVALVES".ST2.SWORD_SLIDE_OUT.in.move_idle ,
         in_sensor_hp1               := I150.1 ,
         in_sensor_hp2               := I150.1 ,
         in_sensor_wp1               := I151.1 ,
         in_sensor_wp2               := I151.1 ,
         out_in_hp                   := "A-DBVALVES".ST2.SWORD_SLIDE_OUT.out.in_hp ,
         out_in_wp                   := "A-DBVALVES".ST2.SWORD_SLIDE_OUT.out.in_wp ,
         out_idle                    := "A-DBVALVES".ST2.SWORD_SLIDE_OUT.out.in_idle ,
         out_status                  := "A-DBVALVES".ST2.SWORD_SLIDE_OUT.out.status ,
         out_brake                   := #brake ,
         out_alarm_hp                := "A-DBVALVES".ST2.SWORD_SLIDE_OUT.out.alarm_hp ,
         out_alarm_wp                := "A-DBVALVES".ST2.SWORD_SLIDE_OUT.out.alarm_wp ,
         out_diag_status             := "A-DBVALVES".ST2.SWORD_SLIDE_OUT.out.diag_status ,
         in_ez_hp                    := Q150.6 ,
         in_ez_wp                    := Q151.6 ,
         in_ez_idle                  := Q1.1
      );

      CALL "3STATE_DIAG"
      (  in_diag_status              := "A-DBVALVES".ST2.SWORD_SLIDE_OUT.out.diag_status ,
         in_Ipw1                     := 'I150.1' ,
         in_Ipw2                     := ' ' ,
         in_Ipr1                     := 'I151.1' ,
         in_Ipr2                     := ' ' ,
         in_Qpw                      := 'Q150.6' ,
         in_Qpr                      := 'Q151.6' ,
         in_tio                      := "A-DBVALVES".io[20]
      );

      A "A-DBVALVES".ST2.SWORD_SLIDE_OUT.out.alarm_hp;
      = "A-ALARMS".VALVES.err2.%X2;

      A "A-DBVALVES".ST2.SWORD_SLIDE_OUT.out.alarm_wp;
      = "A-ALARMS".VALVES.err2.%X3;

      CALL "A-TESTSCL"
      (  in_nr                       := 20 ,
         out                         := "A-DBVALVES".ST2.SWORD_SLIDE_OUT.test
      );

      A(;
      L "A-Doku_DB_OP".HMI.Manual_Functions;
      L 20;
      <>I;
      );
      R "A-DBVALVES".ST2.SWORD_SLIDE_OUT.test.fp_HP;
      R "A-DBVALVES".ST2.SWORD_SLIDE_OUT.test.fp_WP;
      R "A-DBVALVES".ST2.SWORD_SLIDE_OUT.test.fp_IDLE;
NETWORK
TITLE = -

NETWORK
TITLE = [21] ST2 MIECZ - HP
//[21] ST2 SWORD - HP
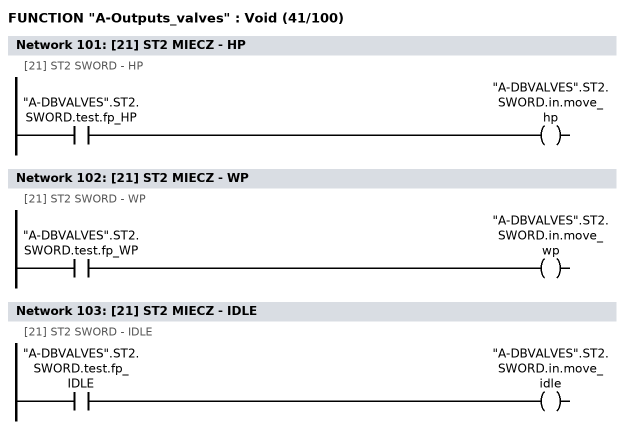
      O "A-DBVALVES".ST2.SWORD.test.fp_HP;
//    O     "A-Flags".STATION.IN_HP_STEP
      = "A-DBVALVES".ST2.SWORD.in.move_hp;
NETWORK
TITLE = [21] ST2 MIECZ - WP
//[21] ST2 SWORD - WP
      O "A-DBVALVES".ST2.SWORD.test.fp_WP;
      = "A-DBVALVES".ST2.SWORD.in.move_wp;
NETWORK
TITLE = [21] ST2 MIECZ - IDLE
//[21] ST2 SWORD - IDLE
      O "A-DBVALVES".ST2.SWORD.test.fp_IDLE;
      = "A-DBVALVES".ST2.SWORD.in.move_idle;
NETWORK
TITLE = [21] ST2 MIECZ
//[21] ST2 SWORD
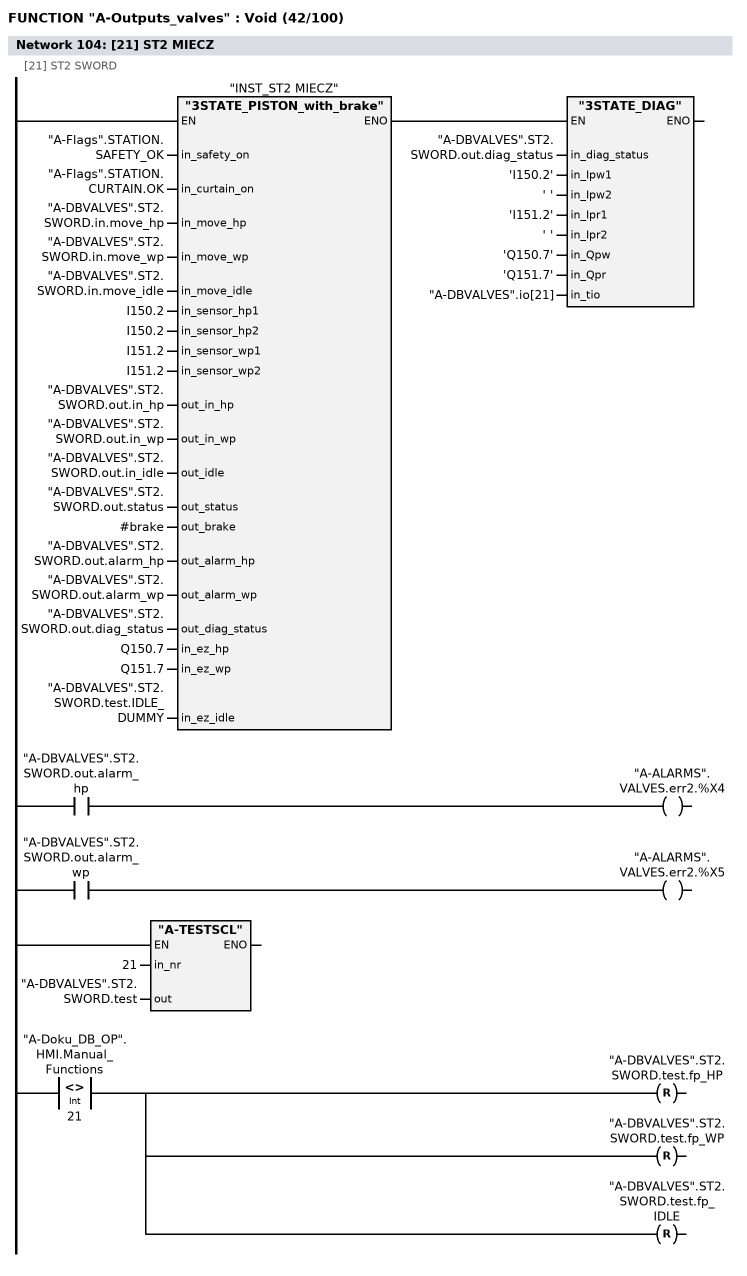
      CALL "3STATE_PISTON_with_brake", "INST_ST2 MIECZ"
      (  in_safety_on                := "A-Flags".STATION.SAFETY_OK ,
         in_curtain_on               := "A-Flags".STATION.CURTAIN.OK ,
         in_move_hp                  := "A-DBVALVES".ST2.SWORD.in.move_hp ,
         in_move_wp                  := "A-DBVALVES".ST2.SWORD.in.move_wp ,
         in_move_idle                := "A-DBVALVES".ST2.SWORD.in.move_idle ,
         in_sensor_hp1               := I150.2 ,
         in_sensor_hp2               := I150.2 ,
         in_sensor_wp1               := I151.2 ,
         in_sensor_wp2               := I151.2 ,
         out_in_hp                   := "A-DBVALVES".ST2.SWORD.out.in_hp ,
         out_in_wp                   := "A-DBVALVES".ST2.SWORD.out.in_wp ,
         out_idle                    := "A-DBVALVES".ST2.SWORD.out.in_idle ,
         out_status                  := "A-DBVALVES".ST2.SWORD.out.status ,
         out_brake                   := #brake ,
         out_alarm_hp                := "A-DBVALVES".ST2.SWORD.out.alarm_hp ,
         out_alarm_wp                := "A-DBVALVES".ST2.SWORD.out.alarm_wp ,
         out_diag_status             := "A-DBVALVES".ST2.SWORD.out.diag_status ,
         in_ez_hp                    := Q150.7 ,
         in_ez_wp                    := Q151.7 ,
         in_ez_idle                  := "A-DBVALVES".ST2.SWORD.test.IDLE_DUMMY
      );

      CALL "3STATE_DIAG"
      (  in_diag_status              := "A-DBVALVES".ST2.SWORD.out.diag_status ,
         in_Ipw1                     := 'I150.2' ,
         in_Ipw2                     := ' ' ,
         in_Ipr1                     := 'I151.2' ,
         in_Ipr2                     := ' ' ,
         in_Qpw                      := 'Q150.7' ,
         in_Qpr                      := 'Q151.7' ,
         in_tio                      := "A-DBVALVES".io[21]
      );

      A "A-DBVALVES".ST2.SWORD.out.alarm_hp;
      = "A-ALARMS".VALVES.err2.%X4;

      A "A-DBVALVES".ST2.SWORD.out.alarm_wp;
      = "A-ALARMS".VALVES.err2.%X5;

      CALL "A-TESTSCL"
      (  in_nr                       := 21 ,
         out                         := "A-DBVALVES".ST2.SWORD.test
      );

      A(;
      L "A-Doku_DB_OP".HMI.Manual_Functions;
      L 21;
      <>I;
      );
      R "A-DBVALVES".ST2.SWORD.test.fp_HP;
      R "A-DBVALVES".ST2.SWORD.test.fp_WP;
      R "A-DBVALVES".ST2.SWORD.test.fp_IDLE;
NETWORK
TITLE = -

NETWORK
TITLE = [22] ST3 MIECZ - HP
//[22] ST3 SWORD - HP
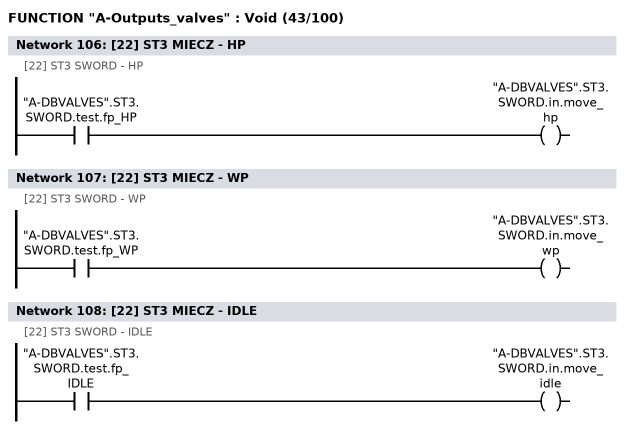
      O "A-DBVALVES".ST3.SWORD.test.fp_HP;
//    O     "A-Flags".STATION.IN_HP_STEP
      = "A-DBVALVES".ST3.SWORD.in.move_hp;
NETWORK
TITLE = [22] ST3 MIECZ - WP
//[22] ST3 SWORD - WP
      O "A-DBVALVES".ST3.SWORD.test.fp_WP;
      = "A-DBVALVES".ST3.SWORD.in.move_wp;
NETWORK
TITLE = [22] ST3 MIECZ - IDLE
//[22] ST3 SWORD - IDLE
      O "A-DBVALVES".ST3.SWORD.test.fp_IDLE;
      = "A-DBVALVES".ST3.SWORD.in.move_idle;
NETWORK
TITLE = [22] ST3 MIECZ
//[22] ST3 SWORD
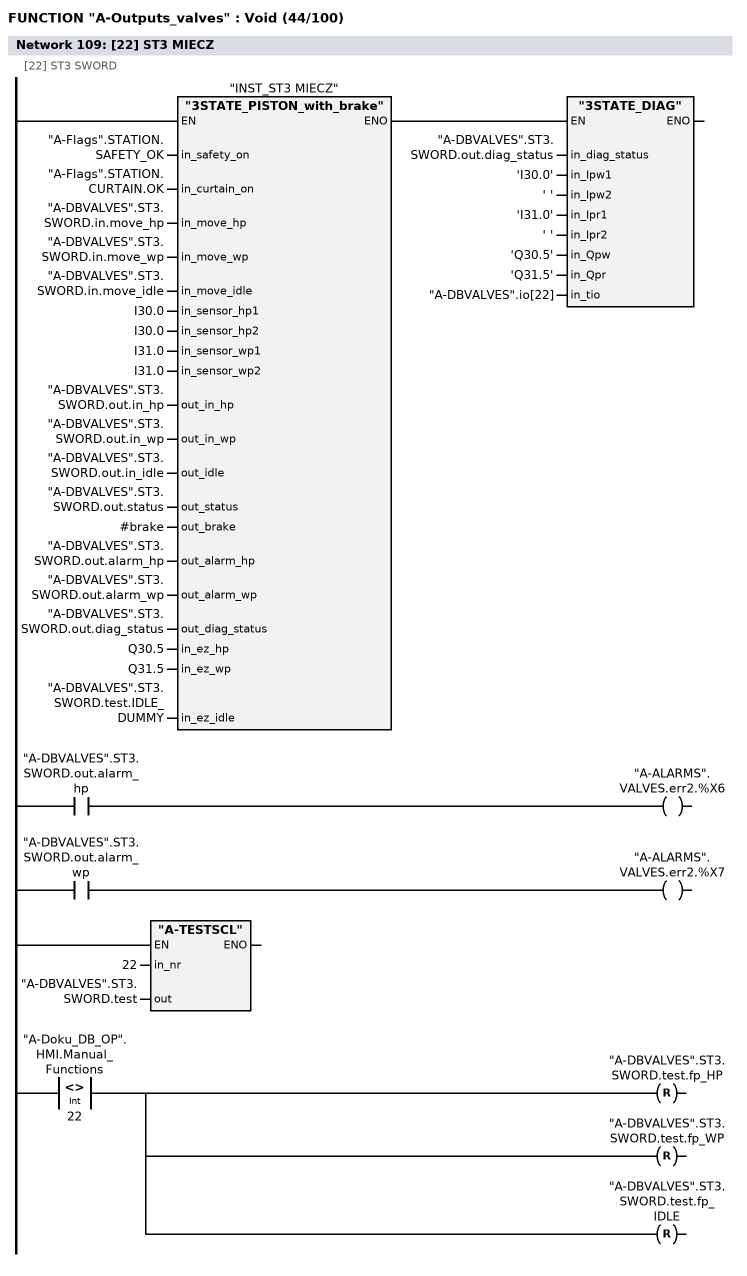
      CALL "3STATE_PISTON_with_brake", "INST_ST3 MIECZ"
      (  in_safety_on                := "A-Flags".STATION.SAFETY_OK ,
         in_curtain_on               := "A-Flags".STATION.CURTAIN.OK ,
         in_move_hp                  := "A-DBVALVES".ST3.SWORD.in.move_hp ,
         in_move_wp                  := "A-DBVALVES".ST3.SWORD.in.move_wp ,
         in_move_idle                := "A-DBVALVES".ST3.SWORD.in.move_idle ,
         in_sensor_hp1               := I30.0 ,
         in_sensor_hp2               := I30.0 ,
         in_sensor_wp1               := I31.0 ,
         in_sensor_wp2               := I31.0 ,
         out_in_hp                   := "A-DBVALVES".ST3.SWORD.out.in_hp ,
         out_in_wp                   := "A-DBVALVES".ST3.SWORD.out.in_wp ,
         out_idle                    := "A-DBVALVES".ST3.SWORD.out.in_idle ,
         out_status                  := "A-DBVALVES".ST3.SWORD.out.status ,
         out_brake                   := #brake ,
         out_alarm_hp                := "A-DBVALVES".ST3.SWORD.out.alarm_hp ,
         out_alarm_wp                := "A-DBVALVES".ST3.SWORD.out.alarm_wp ,
         out_diag_status             := "A-DBVALVES".ST3.SWORD.out.diag_status ,
         in_ez_hp                    := Q30.5 ,
         in_ez_wp                    := Q31.5 ,
         in_ez_idle                  := "A-DBVALVES".ST3.SWORD.test.IDLE_DUMMY
      );

      CALL "3STATE_DIAG"
      (  in_diag_status              := "A-DBVALVES".ST3.SWORD.out.diag_status ,
         in_Ipw1                     := 'I30.0' ,
         in_Ipw2                     := ' ' ,
         in_Ipr1                     := 'I31.0' ,
         in_Ipr2                     := ' ' ,
         in_Qpw                      := 'Q30.5' ,
         in_Qpr                      := 'Q31.5' ,
         in_tio                      := "A-DBVALVES".io[22]
      );

      A "A-DBVALVES".ST3.SWORD.out.alarm_hp;
      = "A-ALARMS".VALVES.err2.%X6;

      A "A-DBVALVES".ST3.SWORD.out.alarm_wp;
      = "A-ALARMS".VALVES.err2.%X7;

      CALL "A-TESTSCL"
      (  in_nr                       := 22 ,
         out                         := "A-DBVALVES".ST3.SWORD.test
      );

      A(;
      L "A-Doku_DB_OP".HMI.Manual_Functions;
      L 22;
      <>I;
      );
      R "A-DBVALVES".ST3.SWORD.test.fp_HP;
      R "A-DBVALVES".ST3.SWORD.test.fp_WP;
      R "A-DBVALVES".ST3.SWORD.test.fp_IDLE;
NETWORK
TITLE = -

NETWORK
TITLE = [23] ST3 ZDERZAK - HP
//[23] ST3 BUMPER - HP
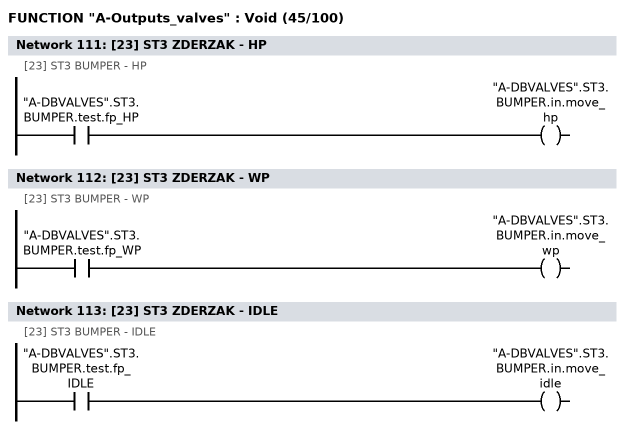
      O "A-DBVALVES".ST3.BUMPER.test.fp_HP;
//    O     "A-Flags".STATION.IN_HP_STEP
      = "A-DBVALVES".ST3.BUMPER.in.move_hp;
NETWORK
TITLE = [23] ST3 ZDERZAK - WP
//[23] ST3 BUMPER - WP
      O "A-DBVALVES".ST3.BUMPER.test.fp_WP;
      = "A-DBVALVES".ST3.BUMPER.in.move_wp;
NETWORK
TITLE = [23] ST3 ZDERZAK - IDLE
//[23] ST3 BUMPER - IDLE
      O "A-DBVALVES".ST3.BUMPER.test.fp_IDLE;
      = "A-DBVALVES".ST3.BUMPER.in.move_idle;
NETWORK
TITLE = [23] ST3 ZDERZAK
//[23] ST3 BUMPER
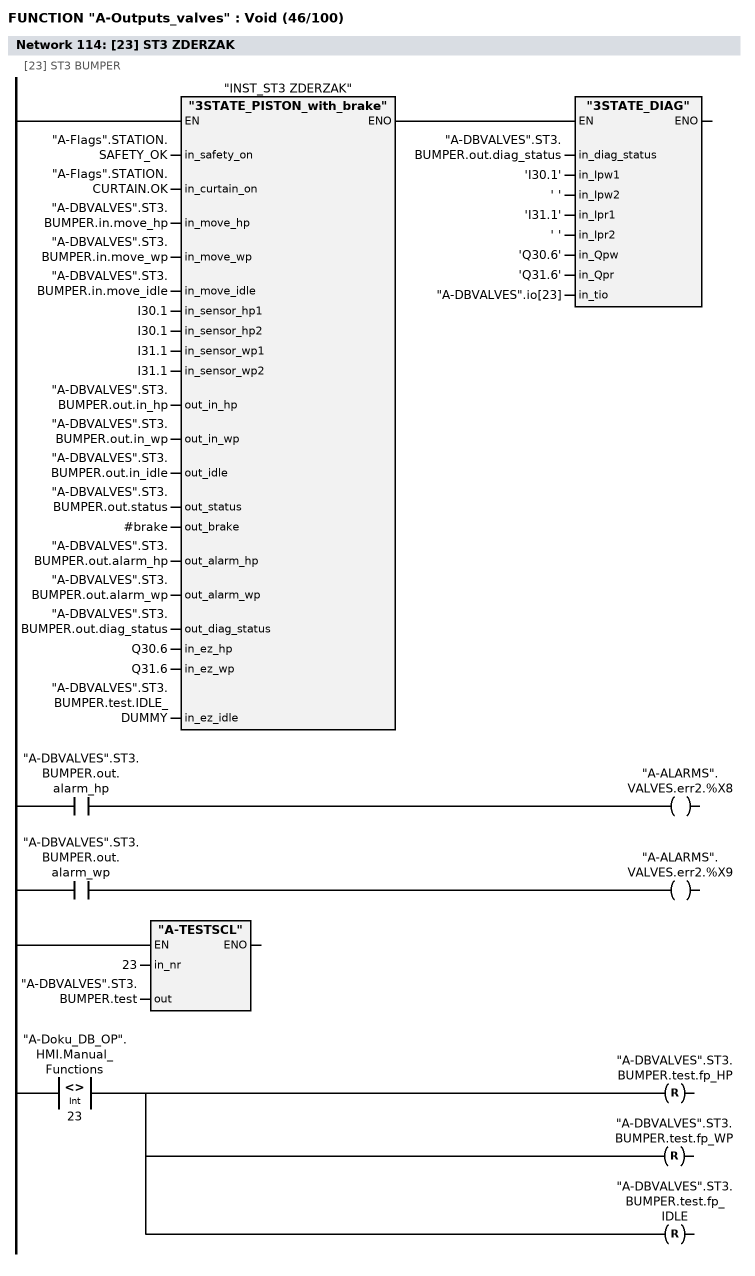
      CALL "3STATE_PISTON_with_brake", "INST_ST3 ZDERZAK"
      (  in_safety_on                := "A-Flags".STATION.SAFETY_OK ,
         in_curtain_on               := "A-Flags".STATION.CURTAIN.OK ,
         in_move_hp                  := "A-DBVALVES".ST3.BUMPER.in.move_hp ,
         in_move_wp                  := "A-DBVALVES".ST3.BUMPER.in.move_wp ,
         in_move_idle                := "A-DBVALVES".ST3.BUMPER.in.move_idle ,
         in_sensor_hp1               := I30.1 ,
         in_sensor_hp2               := I30.1 ,
         in_sensor_wp1               := I31.1 ,
         in_sensor_wp2               := I31.1 ,
         out_in_hp                   := "A-DBVALVES".ST3.BUMPER.out.in_hp ,
         out_in_wp                   := "A-DBVALVES".ST3.BUMPER.out.in_wp ,
         out_idle                    := "A-DBVALVES".ST3.BUMPER.out.in_idle ,
         out_status                  := "A-DBVALVES".ST3.BUMPER.out.status ,
         out_brake                   := #brake ,
         out_alarm_hp                := "A-DBVALVES".ST3.BUMPER.out.alarm_hp ,
         out_alarm_wp                := "A-DBVALVES".ST3.BUMPER.out.alarm_wp ,
         out_diag_status             := "A-DBVALVES".ST3.BUMPER.out.diag_status ,
         in_ez_hp                    := Q30.6 ,
         in_ez_wp                    := Q31.6 ,
         in_ez_idle                  := "A-DBVALVES".ST3.BUMPER.test.IDLE_DUMMY
      );

      CALL "3STATE_DIAG"
      (  in_diag_status              := "A-DBVALVES".ST3.BUMPER.out.diag_status ,
         in_Ipw1                     := 'I30.1' ,
         in_Ipw2                     := ' ' ,
         in_Ipr1                     := 'I31.1' ,
         in_Ipr2                     := ' ' ,
         in_Qpw                      := 'Q30.6' ,
         in_Qpr                      := 'Q31.6' ,
         in_tio                      := "A-DBVALVES".io[23]
      );

      A "A-DBVALVES".ST3.BUMPER.out.alarm_hp;
      = "A-ALARMS".VALVES.err2.%X8;

      A "A-DBVALVES".ST3.BUMPER.out.alarm_wp;
      = "A-ALARMS".VALVES.err2.%X9;

      CALL "A-TESTSCL"
      (  in_nr                       := 23 ,
         out                         := "A-DBVALVES".ST3.BUMPER.test
      );

      A(;
      L "A-Doku_DB_OP".HMI.Manual_Functions;
      L 23;
      <>I;
      );
      R "A-DBVALVES".ST3.BUMPER.test.fp_HP;
      R "A-DBVALVES".ST3.BUMPER.test.fp_WP;
      R "A-DBVALVES".ST3.BUMPER.test.fp_IDLE;
NETWORK
TITLE = -

NETWORK
TITLE = [24] ST3 PODNOSZENIE_MIECZA - HP
//[24] ST3 SWORD_RISING - HP
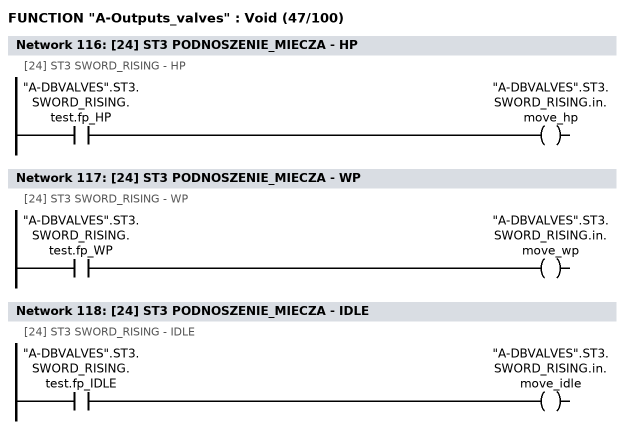
      O "A-DBVALVES".ST3.SWORD_RISING.test.fp_HP;
//    O     "A-Flags".STATION.IN_HP_STEP
      = "A-DBVALVES".ST3.SWORD_RISING.in.move_hp;
NETWORK
TITLE = [24] ST3 PODNOSZENIE_MIECZA - WP
//[24] ST3 SWORD_RISING - WP
      O "A-DBVALVES".ST3.SWORD_RISING.test.fp_WP;
      = "A-DBVALVES".ST3.SWORD_RISING.in.move_wp;
NETWORK
TITLE = [24] ST3 PODNOSZENIE_MIECZA - IDLE
//[24] ST3 SWORD_RISING - IDLE
      O "A-DBVALVES".ST3.SWORD_RISING.test.fp_IDLE;
      = "A-DBVALVES".ST3.SWORD_RISING.in.move_idle;
NETWORK
TITLE = [24] ST3 PODNOSZENIE_MIECZA
//[24] ST3 SWORD_RISING
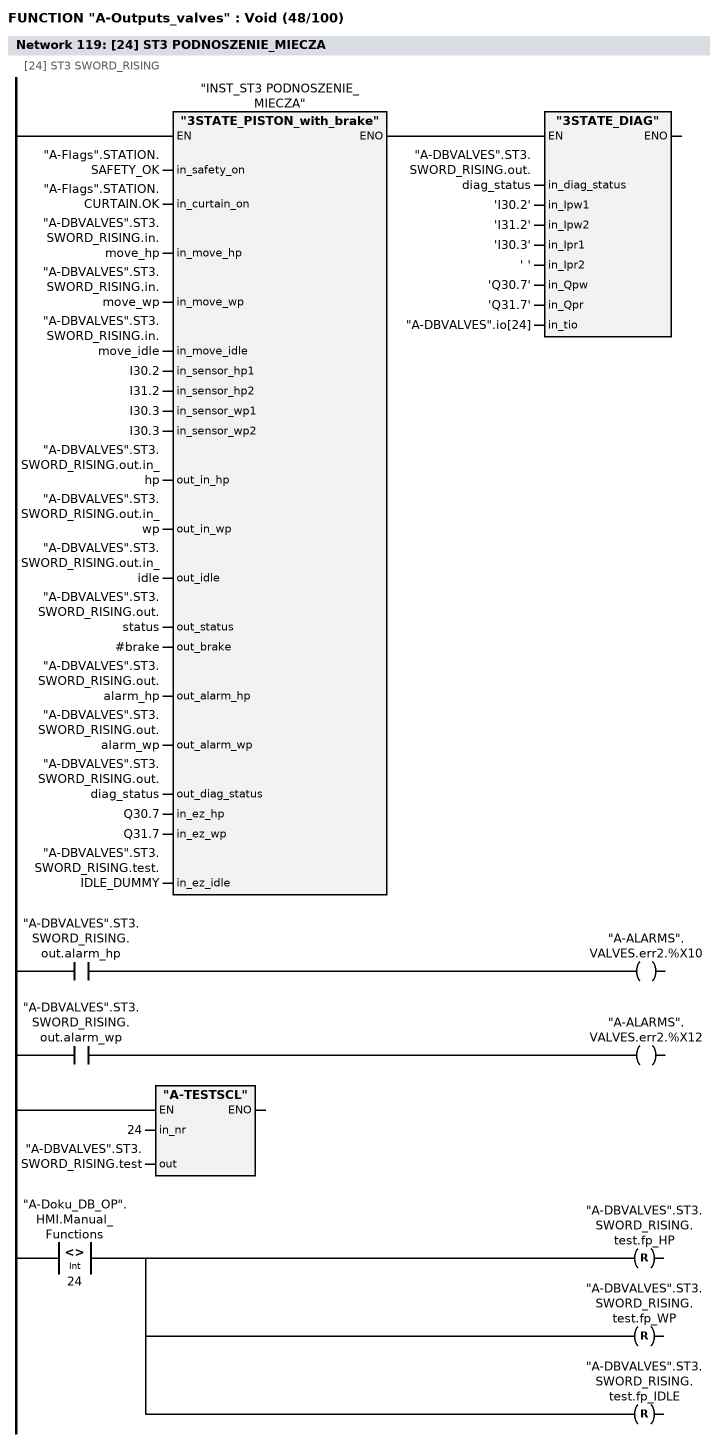
      CALL "3STATE_PISTON_with_brake", "INST_ST3 PODNOSZENIE_MIECZA"
      (  in_safety_on                := "A-Flags".STATION.SAFETY_OK ,
         in_curtain_on               := "A-Flags".STATION.CURTAIN.OK ,
         in_move_hp                  := "A-DBVALVES".ST3.SWORD_RISING.in.move_hp ,
         in_move_wp                  := "A-DBVALVES".ST3.SWORD_RISING.in.move_wp ,
         in_move_idle                := "A-DBVALVES".ST3.SWORD_RISING.in.move_idle ,
         in_sensor_hp1               := I30.2 ,
         in_sensor_hp2               := I31.2 ,
         in_sensor_wp1               := I30.3 ,
         in_sensor_wp2               := I30.3 ,
         out_in_hp                   := "A-DBVALVES".ST3.SWORD_RISING.out.in_hp ,
         out_in_wp                   := "A-DBVALVES".ST3.SWORD_RISING.out.in_wp ,
         out_idle                    := "A-DBVALVES".ST3.SWORD_RISING.out.in_idle ,
         out_status                  := "A-DBVALVES".ST3.SWORD_RISING.out.status ,
         out_brake                   := #brake ,
         out_alarm_hp                := "A-DBVALVES".ST3.SWORD_RISING.out.alarm_hp ,
         out_alarm_wp                := "A-DBVALVES".ST3.SWORD_RISING.out.alarm_wp ,
         out_diag_status             := "A-DBVALVES".ST3.SWORD_RISING.out.diag_status ,
         in_ez_hp                    := Q30.7 ,
         in_ez_wp                    := Q31.7 ,
         in_ez_idle                  := "A-DBVALVES".ST3.SWORD_RISING.test.IDLE_DUMMY
      );

      CALL "3STATE_DIAG"
      (  in_diag_status              := "A-DBVALVES".ST3.SWORD_RISING.out.diag_status ,
         in_Ipw1                     := 'I30.2' ,
         in_Ipw2                     := 'I31.2' ,
         in_Ipr1                     := 'I30.3' ,
         in_Ipr2                     := ' ' ,
         in_Qpw                      := 'Q30.7' ,
         in_Qpr                      := 'Q31.7' ,
         in_tio                      := "A-DBVALVES".io[24]
      );

      A "A-DBVALVES".ST3.SWORD_RISING.out.alarm_hp;
      = "A-ALARMS".VALVES.err2.%X10;

      A "A-DBVALVES".ST3.SWORD_RISING.out.alarm_wp;
      = "A-ALARMS".VALVES.err2.%X12;

      CALL "A-TESTSCL"
      (  in_nr                       := 24 ,
         out                         := "A-DBVALVES".ST3.SWORD_RISING.test
      );

      A(;
      L "A-Doku_DB_OP".HMI.Manual_Functions;
      L 24;
      <>I;
      );
      R "A-DBVALVES".ST3.SWORD_RISING.test.fp_HP;
      R "A-DBVALVES".ST3.SWORD_RISING.test.fp_WP;
      R "A-DBVALVES".ST3.SWORD_RISING.test.fp_IDLE;
NETWORK
TITLE = -

NETWORK
TITLE = [25] ST4 MIECZ - HP
//[25] ST4 SWORD - HP
